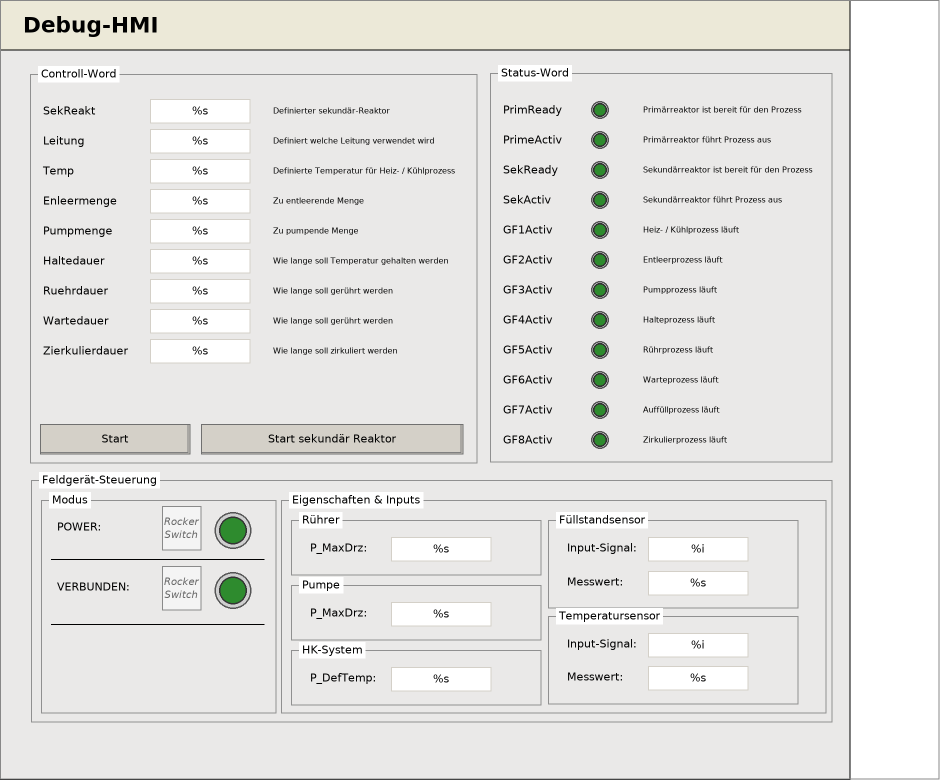
VISUALIZATION Debug_Visu  // 940x780
    Rectangle (0,0 850x780)
    Rectangle (0,0 850x50)
    Label (20,0 830x50), "Debug-HMI"
    GroupBox (30,66 447x397), "Controll-Word"
        Label (10,30 150x30), "SekReakt"
        Label (10,60 150x30), "Leitung"
        Label (10,90 150x30), "Temp"
        Label (10,120 150x30), "Enleermenge"
        Label (10,150 150x30), "Pumpmenge"
        Label (10,180 150x30), "Haltedauer"
        Label (10,210 150x30), "Ruehrdauer"
        Label (10,240 150x30), "Wartedauer"
        Label (10,270 150x30), "Zierkulierdauer"
        Textfield (120,33 100x24), "%s", text variable: MAIN.CW.SekReakt
            OnMouseClick: write MAIN.CW.SekReakt via Edit
        Textfield (120,63 100x24), "%s", text variable: MAIN.CW.Leitung
            OnMouseClick: write MAIN.CW.Leitung via Edit
        Textfield (120,93 100x24), "%s", text variable: MAIN.CW.Temp
            OnMouseClick: write MAIN.CW.Temp via Edit
        Textfield (120,123 100x24), "%s", text variable: MAIN.CW.Enlteermenge
            OnMouseClick: write MAIN.CW.Enlteermenge via Edit
        Textfield (120,153 100x24), "%s", text variable: MAIN.CW.Pumpmenge
            OnMouseClick: write MAIN.CW.Pumpmenge via Edit
        Textfield (120,183 100x24), "%s", text variable: MAIN.CW.Haltedauer
            OnMouseClick: write MAIN.CW.Haltedauer via Edit
        Textfield (120,213 100x24), "%s", text variable: MAIN.CW.Ruehrdauer
            OnMouseClick: write MAIN.CW.Ruehrdauer via Edit
        Textfield (120,243 100x24), "%s", text variable: MAIN.CW.Wartedauer
            OnMouseClick: write MAIN.CW.Wartedauer via Edit
        Textfield (120,273 100x24), "%s", text variable: MAIN.CW.Zirkulierdauer
            OnMouseClick: write MAIN.CW.Zirkulierdauer via Edit
        Label (240,30 300x30), "Definierter sekundär-Reaktor"
        Label (240,60 300x30), "Definiert welche Leitung verwendet wird"
        Label (240,90 300x30), "Definierte Temperatur für Heiz- / Kühlprozess"
        Label (240,120 300x30), "Zu entleerende Menge"
        Label (240,150 300x30), "Zu pumpende Menge"
        Label (240,180 300x30), "Wie lange soll Temperatur gehalten werden"
        Label (240,210 300x30), "Wie lange soll gerührt werden"
        Label (240,240 300x30), "Wie lange soll gerührt werden"
        Label (240,270 300x30), "Wie lange soll zirkuliert werden"
        Button (10,358 150x30), "Start"
            tap GVL.Debug_Start
        Button (171,358 262x30), "Start sekundär Reaktor"
            toggle GVL.Debug_SekStart
    GroupBox (490,65 342x397), "Status-Word"
        Label (10,30 150x30), "PrimReady"
        Label (10,60 150x30), "PrimeActiv"
        Label (10,90 150x30), "SekReady"
        Label (10,120 150x30), "SekActiv"
        Label (10,150 150x30), "GF1Activ"
        Label (10,180 150x30), "GF2Activ"
        Label (10,210 150x30), "GF3Activ"
        Label (10,240 150x30), "GF4Activ"
        Label (10,270 150x30), "GF5Activ"
        Label (150,30 300x30), "Primärreaktor ist bereit für den Prozess"
        Label (150,60 300x30), "Primärreaktor führt Prozess aus"
        Label (150,90 300x30), "Sekundärreaktor ist bereit für den Prozess"
        Label (150,120 300x30), "Sekundärreaktor führt Prozess aus"
        Label (150,150 300x30), "Heiz- / Kühlprozess läuft"
        Label (150,180 300x30), "Entleerprozess läuft"
        Label (150,210 300x30), "Pumpprozess läuft"
        Label (150,240 300x30), "Halteprozess läuft"
        Label (150,270 300x30), "Rührprozess läuft"
        Label (10,300 150x30), "GF6Activ"
        Label (10,330 150x30), "GF7Activ"
        Label (10,360 150x30), "GF8Activ"
        Lamp1 (100,35 20x20), variable: MAIN.SW.PrimReady, style: Lamp-Lamp1-Green
        Lamp1 (100,65 20x20), variable: MAIN.SW.PrimActiv, style: Lamp-Lamp1-Green
        Lamp1 (100,95 20x20), variable: MAIN.SW.SekReady, style: Lamp-Lamp1-Green
        Lamp1 (100,125 20x20), variable: MAIN.SW.SekActiv, style: Lamp-Lamp1-Green
        Lamp1 (100,155 20x20), variable: MAIN.SW.GF1Activ, style: Lamp-Lamp1-Green
        Lamp1 (100,185 20x20), variable: MAIN.SW.GF2Activ, style: Lamp-Lamp1-Green
        Lamp1 (100,215 20x20), variable: MAIN.SW.GF3Activ, style: Lamp-Lamp1-Green
        Lamp1 (100,245 20x20), variable: MAIN.SW.GF4Activ, style: Lamp-Lamp1-Green
        Lamp1 (100,275 20x20), variable: MAIN.SW.GF5Activ, style: Lamp-Lamp1-Green
        Lamp1 (100,305 20x20), variable: MAIN.SW.GF6Activ, style: Lamp-Lamp1-Green
        Lamp1 (100,335 20x20), variable: MAIN.SW.GF7Activ, style: Lamp-Lamp1-Green
        Lamp1 (100,365 20x20), variable: MAIN.SW.GF8Activ, style: Lamp-Lamp1-Green
    Label (640,365 300x30), "Warteprozess läuft"
    Label (640,395 300x30), "Auffüllprozess läuft"
    Label (640,425 300x30), "Zirkulierprozess läuft"
    GroupBox (31,472 801x250), "Feldgerät-Steuerung"
        GroupBox (10,20 235x221), "Modus"
            Label (13,20 150x30), "POWER:"
            RockerSwitch (121,14 39x44), variable: GVL.Bedien_Power, behaviour: TOGGLE, style: Switch-RockerSwitch-Gray
            Lamp1 (191,340 23x30), style: Lamp-Lamp1-Green
            Line (10,67) (223,67)
            Lamp1 (171,17 42x43), variable: GVL.Bedien_Power, style: Lamp-Lamp1-Green
            Label (13,80 150x30), "VERBUNDEN:"
            Line (10,132) (223,132)
        GroupBox (250,20 545x221), "Eigenschaften & Inputs"
            GroupBox (10,20 250x63), "Rührer"
                Label (16,21 79x30), "P_MaxDrz:"
                Textfield (100,25 100x24), "%s", text variable: Reaktoreinheit.NC1.V_DrzMax
                    OnMouseClick: write Reaktoreinheit.NC1.V_DrzMax via Edit
            GroupBox (10,85 250x63), "Pumpe"
                Label (16,21 79x30), "P_MaxDrz:"
                Textfield (100,25 100x24), "%s", text variable: Reaktoreinheit.PS1.V_DrzMax
                    OnMouseClick: write Reaktoreinheit.PS1.V_DrzMax via Edit
            GroupBox (267,20 250x96), "Füllstandsensor"
                Label (16,21 79x30), "Input-Signal:"
                Textfield (100,25 100x24), "%i", text variable: MAIN.CW.Zirkulierdauer
                    OnMouseClick: write Reaktoreinheit.F1.I_iSignal via Edit
                Label (16,55 79x30), "Messwert:"
                Textfield (100,59 100x24), "%s", text variable: Reaktoreinheit.F1.Messwert, input disabled if: TRUE
                    OnMouseClick: write MAIN.CW.Zirkulierdauer via Edit
            GroupBox (267,116 250x96), "Temperatursensor"
                Label (16,21 79x30), "Input-Signal:"
                Textfield (100,25 100x24), "%i", text variable: MAIN.CW.Zirkulierdauer
                    OnMouseClick: write MAIN.CW.Zirkulierdauer via Edit
                Label (16,54 79x30), "Messwert:"
        GroupBox (260,170 250x63), "HK-System"
            Label (16,21 79x30), "P_DefTemp:"
            Textfield (100,25 100x24), "%s", text variable: Reaktoreinheit.HKP1.V_DefTemp
                OnMouseClick: write Reaktoreinheit.HKP1.V_DefTemp via Edit
    RockerSwitch (162,566 39x44), variable: GVL.Debug_Verbunden, behaviour: TOGGLE, style: Switch-RockerSwitch-Gray
    Lamp1 (212,569 42x43), variable: GVL.Debug_Verbunden, style: Lamp-Lamp1-Green
    Textfield (648,666 100x24), "%s", text variable: Reaktoreinheit.T1.Messwert, input disabled if: TRUE
        OnMouseClick: write MAIN.CW.Zirkulierdauer via Edit
END_VISUALIZATION

(* stored: Version 1.1.0.1, ProductVersion 3.1.4024.12
   Visu Debug_Visu: Id {7a986ea6-c035-4ae4-8912-39bf6be96f2f} *)
